TYPE ST_AxisInterface :
STRUCT
    Cmd       : ST_AxisCmd;
    Set       : ST_AxisSet;
    Data      : ST_AxisData;
    State     : ST_AxisState;
    Alarm     : ST_AxisAlarm;
    Interlock : ST_AxisInterlock;
END_STRUCT
END_TYPE

(* stored: Version 1.1.0.1, ProductVersion 3.1.4026.18
   DUT ST_AxisInterface: Id {bc384f07-bbf3-4f6c-845f-b9ff7ce0549c} *)
